// TIA Portal V17 export
// export: Created 2023-02-14T02:49:35.0431365Z, ExportSetting WithDefaults, DisplayName Totally Integrated Automation Portal, DisplayVersion V17, DisplayName TIA Portal Openness, DisplayVersion V17, DisplayName TIA Portal Teamcenter Gateway, DisplayVersion V17, DisplayName TIA Portal Version Control Interface, DisplayVersion V17, DisplayName SINAMICS Startdrive Advanced, DisplayVersion V17, DisplayName SINAMICS Startdrive G130, G150, S120, S150, SINAMICS MV, S210, DisplayVersion V17, DisplayName SINAMICS Startdrive G110M, G120, G120C, G120D, G120P, G115D, DisplayVersion V17, DisplayName STEP 7 Professional, DisplayVersion V17, DisplayName STEP 7 Safety, DisplayVersion V17, DisplayName WinCC Professional, DisplayVersion V17
FUNCTION_BLOCK "IO Valve T09 Garlic"   // FB309, LAD
{ S7_Optimized_Access := 'FALSE' }
VERSION : 0.1
// stored: AutoNumber false, IsIECCheckEnabled false, SetENOAutomatically false, UDAEnableTagReadback false
   VAR_INPUT
      lock : Bool;
      Init : Bool;
      testing : Bool;
      Reset : Bool;
   END_VAR
   VAR
      "AV-09.01" { S7_SetPoint := 'True'} : "Valve";   // AUTO BUTTERFLY VALVE INLET PROCESS WATER TO BFT GARLIC T-09.00
      "AV-09.02" { S7_SetPoint := 'True'} : "Valve";   // AUTO BUTTERFLY VALVE CIP SUPPLY TO BFT GARLIC T-09.00
      "AV-09.03" { S7_SetPoint := 'True'} : "Valve";   // AUTO BUTTERFLY VALVE OUTLET PRODUCT FROM BFT GARLIC T-09.00
      "AV-09.04" { S7_SetPoint := 'True'} : "Valve";   // AUTO BUTTERFLY VALVE CIP SUPPLY TO BFT GARLIC T-09.00
      "AV-09.05" { S7_SetPoint := 'True'} : "Valve";   // AUTO BUTTERFLY VALVE CIP SUPPLY TO BFT GARLIC T-09.00
      "AV-09.06" { S7_SetPoint := 'True'} : "Valve";   // AUTO BUTTERFLY VALVE DRAIN MONO PUMP P-09.01
      "AV-09.07" { S7_SetPoint := 'True'} : "Valve";   // AUTO BUTTERFLY VALVE INLET VINEGAR FROM T-10.00 TO BLENDING TANK T-20.00
      "AV-09.08" { S7_SetPoint := 'True'} : "Valve";
      "AV-09.09" { S7_SetPoint := 'True'} : "Valve";
      "AV-09.10" { S7_SetPoint := 'True'} : "Valve";
      "AV-09.11" { S7_SetPoint := 'True'} : "Valve";
      "AV-09.12" { S7_SetPoint := 'True'} : "Valve";
      "AV-09.13" { S7_SetPoint := 'True'} : "Valve";
      "AV-09.14" { S7_SetPoint := 'True'} : "Valve";
      "AV-09.15" { S7_SetPoint := 'True'} : "Valve";
   END_VAR
BEGIN

REGION Network 1 (SCL): FB OPEN and CLOSE
   IF #testing THEN
       // Statement section IF
       #"AV-09.01".FB_OPEN := #"AV-09.01".QCMD_OP;
       #"AV-09.01".FB_CLOSE := NOT #"AV-09.01".QCMD_OP;
       #"AV-09.02".FB_OPEN := #"AV-09.02".QCMD_OP;
       #"AV-09.02".FB_CLOSE := NOT #"AV-09.02".QCMD_OP;
       #"AV-09.03".FB_OPEN := #"AV-09.03".QCMD_OP;
       #"AV-09.03".FB_CLOSE := NOT #"AV-09.03".QCMD_OP;
       #"AV-09.04".FB_OPEN := #"AV-09.04".QCMD_OP;
       #"AV-09.04".FB_CLOSE := NOT #"AV-09.04".QCMD_OP;
       #"AV-09.05".FB_OPEN := #"AV-09.05".QCMD_OP;
       #"AV-09.05".FB_CLOSE := NOT #"AV-09.05".QCMD_OP;
       #"AV-09.06".FB_OPEN := #"AV-09.06".QCMD_OP;
       #"AV-09.06".FB_CLOSE := NOT #"AV-09.06".QCMD_OP;
       #"AV-09.07".FB_OPEN := #"AV-09.07".QCMD_OP;
       #"AV-09.07".FB_CLOSE := NOT #"AV-09.07".QCMD_OP;
       #"AV-09.08".FB_OPEN := #"AV-09.08".QCMD_OP;
       #"AV-09.08".FB_CLOSE := NOT #"AV-09.08".QCMD_OP;
       #"AV-09.09".FB_OPEN := #"AV-09.09".QCMD_OP;
       #"AV-09.09".FB_CLOSE := NOT #"AV-09.09".QCMD_OP;
       #"AV-09.10".FB_OPEN := #"AV-09.10".QCMD_OP;
       #"AV-09.10".FB_CLOSE := NOT #"AV-09.10".QCMD_OP;
       #"AV-09.11".FB_OPEN := #"AV-09.11".QCMD_OP;
       #"AV-09.11".FB_CLOSE := NOT #"AV-09.11".QCMD_OP;
       #"AV-09.12".FB_OPEN := #"AV-09.12".QCMD_OP;
       #"AV-09.12".FB_CLOSE := NOT #"AV-09.12".QCMD_OP;
       #"AV-09.13".FB_OPEN := #"AV-09.13".QCMD_OP;
       #"AV-09.13".FB_CLOSE := NOT #"AV-09.13".QCMD_OP;
       #"AV-09.14".FB_OPEN := #"AV-09.14".QCMD_OP;
       #"AV-09.14".FB_CLOSE := NOT #"AV-09.14".QCMD_OP;
       #"AV-09.15".FB_OPEN := #"AV-09.15".QCMD_OP;
       #"AV-09.15".FB_CLOSE := NOT #"AV-09.15".QCMD_OP;
   ELSE
       // Statement section ELSE
       #"AV-09.01".FB_OPEN := NOT "ZSC-09.01";
       #"AV-09.01".FB_CLOSE := "ZSC-09.01";
       #"AV-09.02".FB_OPEN := NOT "ZSC-09.02";
       #"AV-09.02".FB_CLOSE := "ZSC-09.02";
       #"AV-09.03".FB_OPEN := NOT "ZSC-09.03";
       #"AV-09.03".FB_CLOSE := "ZSC-09.03";
       #"AV-09.04".FB_OPEN := NOT "ZSC-09.04";
       #"AV-09.04".FB_CLOSE := "ZSC-09.04";
       #"AV-09.05".FB_OPEN := NOT "ZSC-09.05";
       #"AV-09.05".FB_CLOSE := "ZSC-09.05";
       #"AV-09.06".FB_OPEN := #"AV-09.06".QCMD_OP;
       #"AV-09.06".FB_CLOSE := NOT #"AV-09.06".QCMD_OP;
       #"AV-09.07".FB_OPEN := #"AV-09.07".QCMD_OP;
       #"AV-09.07".FB_CLOSE := NOT #"AV-09.07".QCMD_OP;
       #"AV-09.08".FB_OPEN := #"AV-09.08".QCMD_OP;
       #"AV-09.08".FB_CLOSE := NOT #"AV-09.08".QCMD_OP;
       #"AV-09.09".FB_OPEN := #"AV-09.09".QCMD_OP;
       #"AV-09.09".FB_CLOSE := NOT #"AV-09.09".QCMD_OP;
       #"AV-09.10".FB_OPEN := #"AV-09.10".QCMD_OP;
       #"AV-09.10".FB_CLOSE := NOT #"AV-09.10".QCMD_OP;
       #"AV-09.11".FB_OPEN := NOT "ZSC-09.11";
       #"AV-09.11".FB_CLOSE := "ZSC-09.11";
       #"AV-09.12".FB_OPEN := NOT "ZSC-09.12";
       #"AV-09.12".FB_CLOSE := "ZSC-09.12";
       #"AV-09.13".FB_OPEN := NOT "ZSC-09.13";
       #"AV-09.13".FB_CLOSE := "ZSC-09.13";
       #"AV-09.14".FB_OPEN := #"AV-09.14".QCMD_OP;
       #"AV-09.14".FB_CLOSE := NOT #"AV-09.14".QCMD_OP;
       #"AV-09.15".FB_OPEN := #"AV-09.15".QCMD_OP;
       #"AV-09.15".FB_CLOSE := NOT #"AV-09.15".QCMD_OP;
   END_IF;
END_REGION

NETWORK
TITLE = FB Monitoring Time
// FB OPEN Time
      L     t#20s;
      T     #"AV-09.01".MON_T;
      T     #"AV-09.02".MON_T;
      T     #"AV-09.03".MON_T;
      T     #"AV-09.04".MON_T;
      T     #"AV-09.05".MON_T;
      T     #"AV-09.06".MON_T;
      T     #"AV-09.07".MON_T;
      T     #"AV-09.08".MON_T;
      T     #"AV-09.09".MON_T;
      T     #"AV-09.10".MON_T;
      T     #"AV-09.11".MON_T;
      T     #"AV-09.12".MON_T;
      T     #"AV-09.13".MON_T;
      T     #"AV-09.14".MON_T;
      T     #"AV-09.15".MON_T;
// FB CLOSE Time
      L     t#20s;
      T     #"AV-09.01".MON_T_CLOSE;
      T     #"AV-09.02".MON_T_CLOSE;
      T     #"AV-09.03".MON_T_CLOSE;
      T     #"AV-09.04".MON_T_CLOSE;
      T     #"AV-09.05".MON_T_CLOSE;
      T     #"AV-09.06".MON_T_CLOSE;
      T     #"AV-09.07".MON_T_CLOSE;
      T     #"AV-09.08".MON_T_CLOSE;
      T     #"AV-09.09".MON_T_CLOSE;
      T     #"AV-09.10".MON_T_CLOSE;
      T     #"AV-09.11".MON_T_CLOSE;
      T     #"AV-09.12".MON_T_CLOSE;
      T     #"AV-09.13".MON_T_CLOSE;
      T     #"AV-09.14".MON_T_CLOSE;
      T     #"AV-09.15".MON_T_CLOSE;

REGION Network 3: AV-09.01 w ZSC
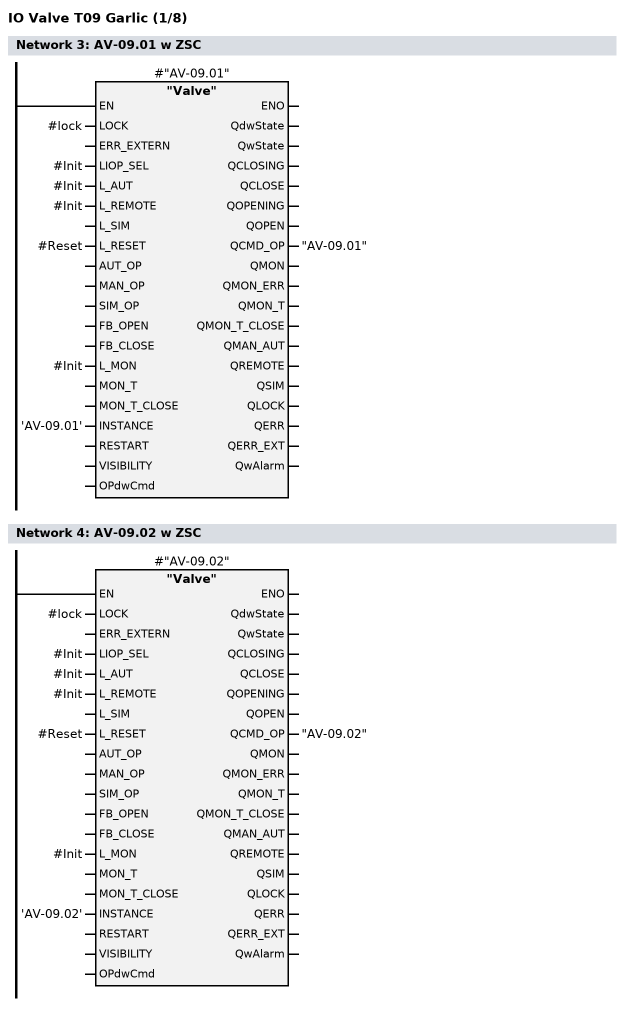
   RUNG wire#powerrail
      #"AV-09.01"(LOCK := #lock, ERR_EXTERN :=, LIOP_SEL := #Init, L_AUT := #Init, L_REMOTE := #Init, L_SIM :=, L_RESET := #Reset, AUT_OP :=, MAN_OP :=, SIM_OP :=, FB_OPEN :=, FB_CLOSE :=, L_MON := #Init, MON_T :=, MON_T_CLOSE :=, INSTANCE := 'AV-09.01', RESTART :=, VISIBILITY :=, OPdwCmd :=, QdwState =>, QwState =>, QCLOSING =>, QCLOSE =>, QOPENING =>, QOPEN =>, QCMD_OP => "AV-09.01", QMON =>, QMON_ERR =>, QMON_T =>, QMON_T_CLOSE =>, QMAN_AUT =>, QREMOTE =>, QSIM =>, QLOCK =>, QERR =>, QERR_EXT =>, QwAlarm =>)
   END_RUNG
   // the same network as SCL:
   #"AV-09.01"(LOCK := #lock,   // "Valve"
               LIOP_SEL := #Init,
               L_AUT := #Init,
               L_REMOTE := #Init,
               L_RESET := #Reset,
               L_MON := #Init,
               INSTANCE := 'AV-09.01',
               QCMD_OP => "AV-09.01");
END_REGION

REGION Network 4: AV-09.02 w ZSC
   RUNG wire#powerrail
      #"AV-09.02"(LOCK := #lock, ERR_EXTERN :=, LIOP_SEL := #Init, L_AUT := #Init, L_REMOTE := #Init, L_SIM :=, L_RESET := #Reset, AUT_OP :=, MAN_OP :=, SIM_OP :=, FB_OPEN :=, FB_CLOSE :=, L_MON := #Init, MON_T :=, MON_T_CLOSE :=, INSTANCE := 'AV-09.02', RESTART :=, VISIBILITY :=, OPdwCmd :=, QdwState =>, QwState =>, QCLOSING =>, QCLOSE =>, QOPENING =>, QOPEN =>, QCMD_OP => "AV-09.02", QMON =>, QMON_ERR =>, QMON_T =>, QMON_T_CLOSE =>, QMAN_AUT =>, QREMOTE =>, QSIM =>, QLOCK =>, QERR =>, QERR_EXT =>, QwAlarm =>)
   END_RUNG
   // the same network as SCL:
   #"AV-09.02"(LOCK := #lock,   // "Valve"
               LIOP_SEL := #Init,
               L_AUT := #Init,
               L_REMOTE := #Init,
               L_RESET := #Reset,
               L_MON := #Init,
               INSTANCE := 'AV-09.02',
               QCMD_OP => "AV-09.02");
END_REGION

REGION Network 5: AV-09.03 w ZSC
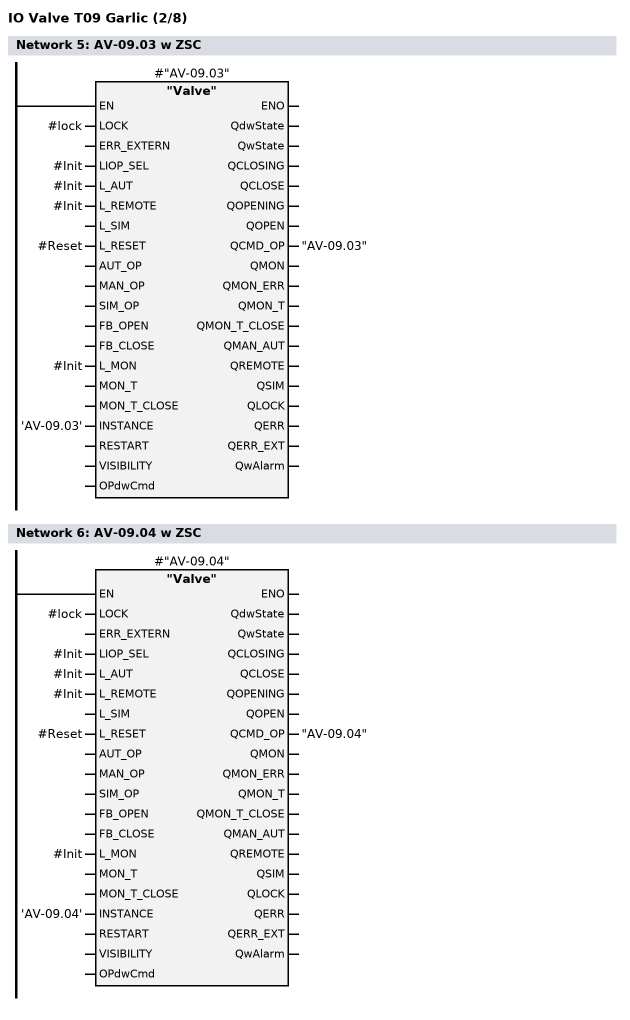
   RUNG wire#powerrail
      #"AV-09.03"(LOCK := #lock, ERR_EXTERN :=, LIOP_SEL := #Init, L_AUT := #Init, L_REMOTE := #Init, L_SIM :=, L_RESET := #Reset, AUT_OP :=, MAN_OP :=, SIM_OP :=, FB_OPEN :=, FB_CLOSE :=, L_MON := #Init, MON_T :=, MON_T_CLOSE :=, INSTANCE := 'AV-09.03', RESTART :=, VISIBILITY :=, OPdwCmd :=, QdwState =>, QwState =>, QCLOSING =>, QCLOSE =>, QOPENING =>, QOPEN =>, QCMD_OP => "AV-09.03", QMON =>, QMON_ERR =>, QMON_T =>, QMON_T_CLOSE =>, QMAN_AUT =>, QREMOTE =>, QSIM =>, QLOCK =>, QERR =>, QERR_EXT =>, QwAlarm =>)
   END_RUNG
   // the same network as SCL:
   #"AV-09.03"(LOCK := #lock,   // "Valve"
               LIOP_SEL := #Init,
               L_AUT := #Init,
               L_REMOTE := #Init,
               L_RESET := #Reset,
               L_MON := #Init,
               INSTANCE := 'AV-09.03',
               QCMD_OP => "AV-09.03");
END_REGION

REGION Network 6: AV-09.04 w ZSC
   RUNG wire#powerrail
      #"AV-09.04"(LOCK := #lock, ERR_EXTERN :=, LIOP_SEL := #Init, L_AUT := #Init, L_REMOTE := #Init, L_SIM :=, L_RESET := #Reset, AUT_OP :=, MAN_OP :=, SIM_OP :=, FB_OPEN :=, FB_CLOSE :=, L_MON := #Init, MON_T :=, MON_T_CLOSE :=, INSTANCE := 'AV-09.04', RESTART :=, VISIBILITY :=, OPdwCmd :=, QdwState =>, QwState =>, QCLOSING =>, QCLOSE =>, QOPENING =>, QOPEN =>, QCMD_OP => "AV-09.04", QMON =>, QMON_ERR =>, QMON_T =>, QMON_T_CLOSE =>, QMAN_AUT =>, QREMOTE =>, QSIM =>, QLOCK =>, QERR =>, QERR_EXT =>, QwAlarm =>)
   END_RUNG
   // the same network as SCL:
   #"AV-09.04"(LOCK := #lock,   // "Valve"
               LIOP_SEL := #Init,
               L_AUT := #Init,
               L_REMOTE := #Init,
               L_RESET := #Reset,
               L_MON := #Init,
               INSTANCE := 'AV-09.04',
               QCMD_OP => "AV-09.04");
END_REGION

REGION Network 7: AV-09.05 w ZSC
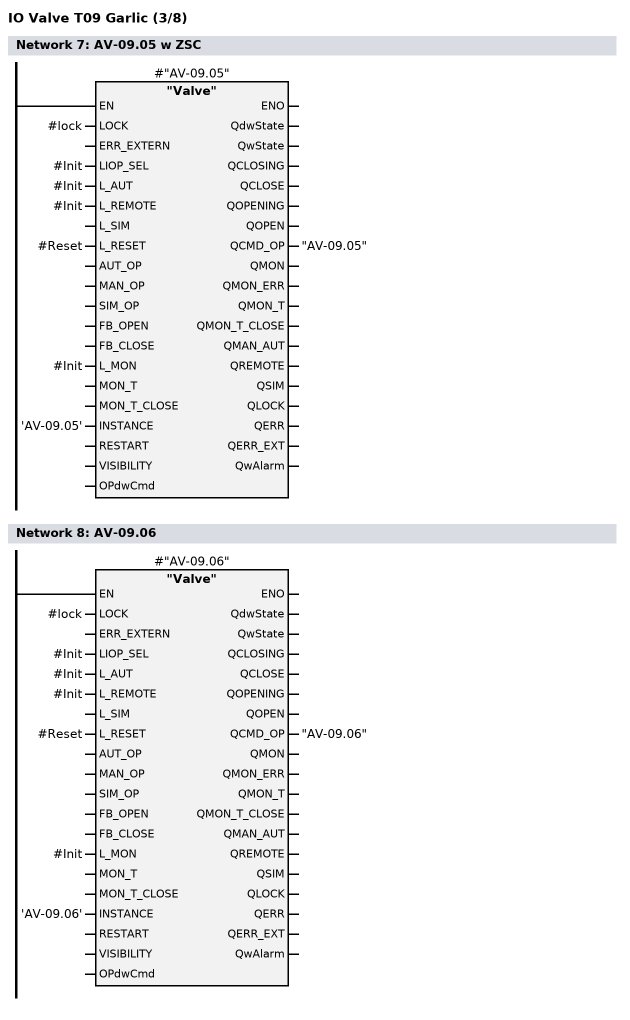
   RUNG wire#powerrail
      #"AV-09.05"(LOCK := #lock, ERR_EXTERN :=, LIOP_SEL := #Init, L_AUT := #Init, L_REMOTE := #Init, L_SIM :=, L_RESET := #Reset, AUT_OP :=, MAN_OP :=, SIM_OP :=, FB_OPEN :=, FB_CLOSE :=, L_MON := #Init, MON_T :=, MON_T_CLOSE :=, INSTANCE := 'AV-09.05', RESTART :=, VISIBILITY :=, OPdwCmd :=, QdwState =>, QwState =>, QCLOSING =>, QCLOSE =>, QOPENING =>, QOPEN =>, QCMD_OP => "AV-09.05", QMON =>, QMON_ERR =>, QMON_T =>, QMON_T_CLOSE =>, QMAN_AUT =>, QREMOTE =>, QSIM =>, QLOCK =>, QERR =>, QERR_EXT =>, QwAlarm =>)
   END_RUNG
   // the same network as SCL:
   #"AV-09.05"(LOCK := #lock,   // "Valve"
               LIOP_SEL := #Init,
               L_AUT := #Init,
               L_REMOTE := #Init,
               L_RESET := #Reset,
               L_MON := #Init,
               INSTANCE := 'AV-09.05',
               QCMD_OP => "AV-09.05");
END_REGION

REGION Network 8: AV-09.06
   RUNG wire#powerrail
      #"AV-09.06"(LOCK := #lock, ERR_EXTERN :=, LIOP_SEL := #Init, L_AUT := #Init, L_REMOTE := #Init, L_SIM :=, L_RESET := #Reset, AUT_OP :=, MAN_OP :=, SIM_OP :=, FB_OPEN :=, FB_CLOSE :=, L_MON := #Init, MON_T :=, MON_T_CLOSE :=, INSTANCE := 'AV-09.06', RESTART :=, VISIBILITY :=, OPdwCmd :=, QdwState =>, QwState =>, QCLOSING =>, QCLOSE =>, QOPENING =>, QOPEN =>, QCMD_OP => "AV-09.06", QMON =>, QMON_ERR =>, QMON_T =>, QMON_T_CLOSE =>, QMAN_AUT =>, QREMOTE =>, QSIM =>, QLOCK =>, QERR =>, QERR_EXT =>, QwAlarm =>)
   END_RUNG
   // the same network as SCL:
   #"AV-09.06"(LOCK := #lock,   // "Valve"
               LIOP_SEL := #Init,
               L_AUT := #Init,
               L_REMOTE := #Init,
               L_RESET := #Reset,
               L_MON := #Init,
               INSTANCE := 'AV-09.06',
               QCMD_OP => "AV-09.06");
END_REGION

REGION Network 9: AV-09.07
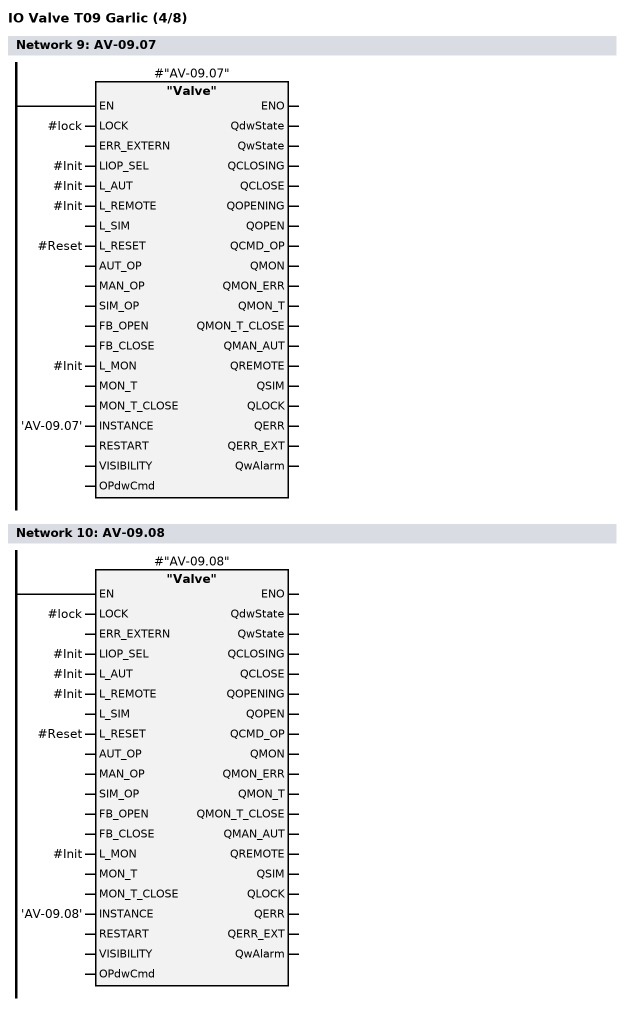
   RUNG wire#powerrail
      #"AV-09.07"(LOCK := #lock, ERR_EXTERN :=, LIOP_SEL := #Init, L_AUT := #Init, L_REMOTE := #Init, L_SIM :=, L_RESET := #Reset, AUT_OP :=, MAN_OP :=, SIM_OP :=, FB_OPEN :=, FB_CLOSE :=, L_MON := #Init, MON_T :=, MON_T_CLOSE :=, INSTANCE := 'AV-09.07', RESTART :=, VISIBILITY :=, OPdwCmd :=, QdwState =>, QwState =>, QCLOSING =>, QCLOSE =>, QOPENING =>, QOPEN =>, QCMD_OP =>, QMON =>, QMON_ERR =>, QMON_T =>, QMON_T_CLOSE =>, QMAN_AUT =>, QREMOTE =>, QSIM =>, QLOCK =>, QERR =>, QERR_EXT =>, QwAlarm =>)
   END_RUNG
   // the same network as SCL:
   #"AV-09.07"(LOCK := #lock,   // "Valve"
               LIOP_SEL := #Init,
               L_AUT := #Init,
               L_REMOTE := #Init,
               L_RESET := #Reset,
               L_MON := #Init,
               INSTANCE := 'AV-09.07');
END_REGION

REGION Network 10: AV-09.08
   RUNG wire#powerrail
      #"AV-09.08"(LOCK := #lock, ERR_EXTERN :=, LIOP_SEL := #Init, L_AUT := #Init, L_REMOTE := #Init, L_SIM :=, L_RESET := #Reset, AUT_OP :=, MAN_OP :=, SIM_OP :=, FB_OPEN :=, FB_CLOSE :=, L_MON := #Init, MON_T :=, MON_T_CLOSE :=, INSTANCE := 'AV-09.08', RESTART :=, VISIBILITY :=, OPdwCmd :=, QdwState =>, QwState =>, QCLOSING =>, QCLOSE =>, QOPENING =>, QOPEN =>, QCMD_OP =>, QMON =>, QMON_ERR =>, QMON_T =>, QMON_T_CLOSE =>, QMAN_AUT =>, QREMOTE =>, QSIM =>, QLOCK =>, QERR =>, QERR_EXT =>, QwAlarm =>)
   END_RUNG
   // the same network as SCL:
   #"AV-09.08"(LOCK := #lock,   // "Valve"
               LIOP_SEL := #Init,
               L_AUT := #Init,
               L_REMOTE := #Init,
               L_RESET := #Reset,
               L_MON := #Init,
               INSTANCE := 'AV-09.08');
END_REGION

REGION Network 11: AV-09.09
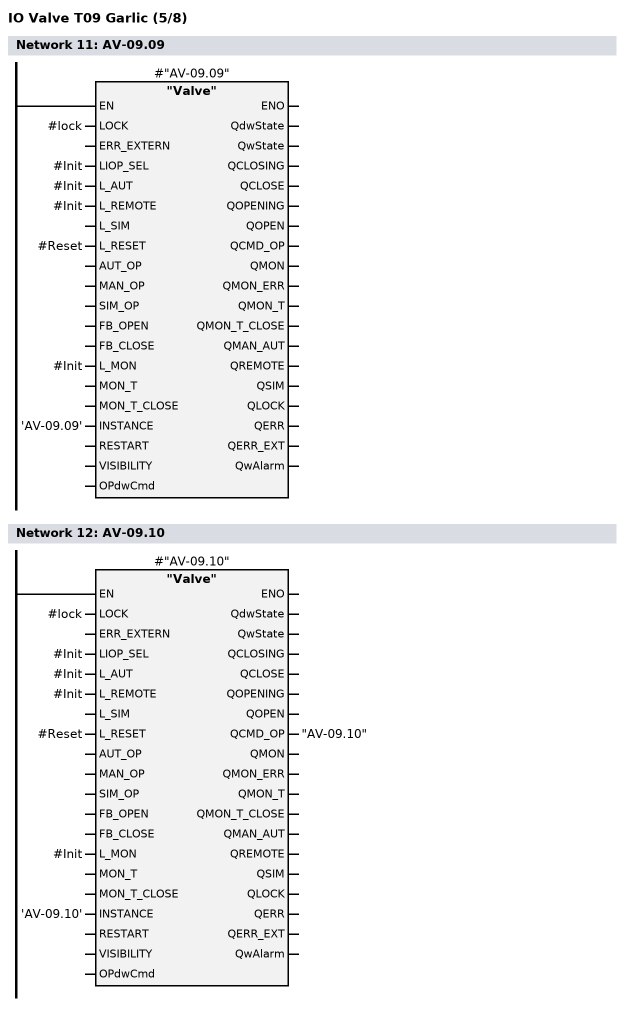
   RUNG wire#powerrail
      #"AV-09.09"(LOCK := #lock, ERR_EXTERN :=, LIOP_SEL := #Init, L_AUT := #Init, L_REMOTE := #Init, L_SIM :=, L_RESET := #Reset, AUT_OP :=, MAN_OP :=, SIM_OP :=, FB_OPEN :=, FB_CLOSE :=, L_MON := #Init, MON_T :=, MON_T_CLOSE :=, INSTANCE := 'AV-09.09', RESTART :=, VISIBILITY :=, OPdwCmd :=, QdwState =>, QwState =>, QCLOSING =>, QCLOSE =>, QOPENING =>, QOPEN =>, QCMD_OP =>, QMON =>, QMON_ERR =>, QMON_T =>, QMON_T_CLOSE =>, QMAN_AUT =>, QREMOTE =>, QSIM =>, QLOCK =>, QERR =>, QERR_EXT =>, QwAlarm =>)
   END_RUNG
   // the same network as SCL:
   #"AV-09.09"(LOCK := #lock,   // "Valve"
               LIOP_SEL := #Init,
               L_AUT := #Init,
               L_REMOTE := #Init,
               L_RESET := #Reset,
               L_MON := #Init,
               INSTANCE := 'AV-09.09');
END_REGION

REGION Network 12: AV-09.10
   RUNG wire#powerrail
      #"AV-09.10"(LOCK := #lock, ERR_EXTERN :=, LIOP_SEL := #Init, L_AUT := #Init, L_REMOTE := #Init, L_SIM :=, L_RESET := #Reset, AUT_OP :=, MAN_OP :=, SIM_OP :=, FB_OPEN :=, FB_CLOSE :=, L_MON := #Init, MON_T :=, MON_T_CLOSE :=, INSTANCE := 'AV-09.10', RESTART :=, VISIBILITY :=, OPdwCmd :=, QdwState =>, QwState =>, QCLOSING =>, QCLOSE =>, QOPENING =>, QOPEN =>, QCMD_OP => "AV-09.10", QMON =>, QMON_ERR =>, QMON_T =>, QMON_T_CLOSE =>, QMAN_AUT =>, QREMOTE =>, QSIM =>, QLOCK =>, QERR =>, QERR_EXT =>, QwAlarm =>)
   END_RUNG
   // the same network as SCL:
   #"AV-09.10"(LOCK := #lock,   // "Valve"
               LIOP_SEL := #Init,
               L_AUT := #Init,
               L_REMOTE := #Init,
               L_RESET := #Reset,
               L_MON := #Init,
               INSTANCE := 'AV-09.10',
               QCMD_OP => "AV-09.10");
END_REGION

REGION Network 13: AV-09.11 w ZSC
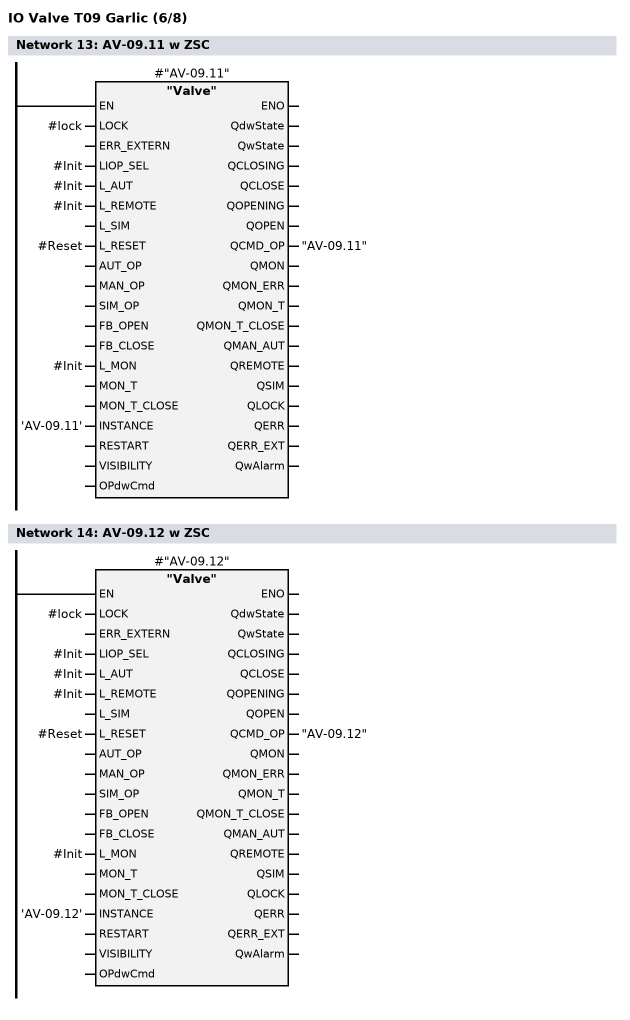
   RUNG wire#powerrail
      #"AV-09.11"(LOCK := #lock, ERR_EXTERN :=, LIOP_SEL := #Init, L_AUT := #Init, L_REMOTE := #Init, L_SIM :=, L_RESET := #Reset, AUT_OP :=, MAN_OP :=, SIM_OP :=, FB_OPEN :=, FB_CLOSE :=, L_MON := #Init, MON_T :=, MON_T_CLOSE :=, INSTANCE := 'AV-09.11', RESTART :=, VISIBILITY :=, OPdwCmd :=, QdwState =>, QwState =>, QCLOSING =>, QCLOSE =>, QOPENING =>, QOPEN =>, QCMD_OP => "AV-09.11", QMON =>, QMON_ERR =>, QMON_T =>, QMON_T_CLOSE =>, QMAN_AUT =>, QREMOTE =>, QSIM =>, QLOCK =>, QERR =>, QERR_EXT =>, QwAlarm =>)
   END_RUNG
   // the same network as SCL:
   #"AV-09.11"(LOCK := #lock,   // "Valve"
               LIOP_SEL := #Init,
               L_AUT := #Init,
               L_REMOTE := #Init,
               L_RESET := #Reset,
               L_MON := #Init,
               INSTANCE := 'AV-09.11',
               QCMD_OP => "AV-09.11");
END_REGION

REGION Network 14: AV-09.12 w ZSC
   RUNG wire#powerrail
      #"AV-09.12"(LOCK := #lock, ERR_EXTERN :=, LIOP_SEL := #Init, L_AUT := #Init, L_REMOTE := #Init, L_SIM :=, L_RESET := #Reset, AUT_OP :=, MAN_OP :=, SIM_OP :=, FB_OPEN :=, FB_CLOSE :=, L_MON := #Init, MON_T :=, MON_T_CLOSE :=, INSTANCE := 'AV-09.12', RESTART :=, VISIBILITY :=, OPdwCmd :=, QdwState =>, QwState =>, QCLOSING =>, QCLOSE =>, QOPENING =>, QOPEN =>, QCMD_OP => "AV-09.12", QMON =>, QMON_ERR =>, QMON_T =>, QMON_T_CLOSE =>, QMAN_AUT =>, QREMOTE =>, QSIM =>, QLOCK =>, QERR =>, QERR_EXT =>, QwAlarm =>)
   END_RUNG
   // the same network as SCL:
   #"AV-09.12"(LOCK := #lock,   // "Valve"
               LIOP_SEL := #Init,
               L_AUT := #Init,
               L_REMOTE := #Init,
               L_RESET := #Reset,
               L_MON := #Init,
               INSTANCE := 'AV-09.12',
               QCMD_OP => "AV-09.12");
END_REGION

REGION Network 15: AV-09.13 w ZSC
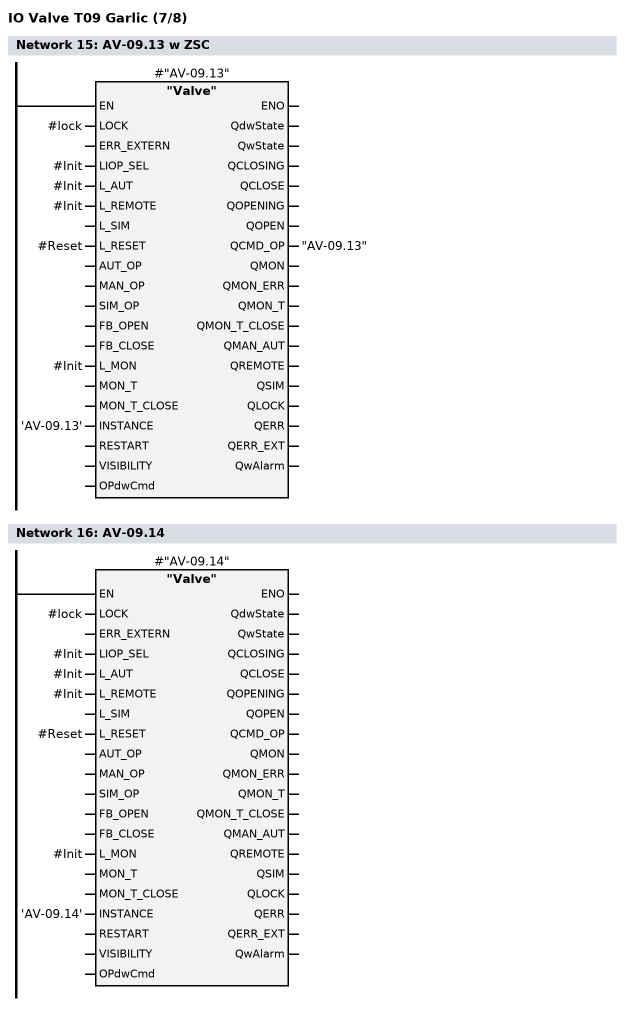
   RUNG wire#powerrail
      #"AV-09.13"(LOCK := #lock, ERR_EXTERN :=, LIOP_SEL := #Init, L_AUT := #Init, L_REMOTE := #Init, L_SIM :=, L_RESET := #Reset, AUT_OP :=, MAN_OP :=, SIM_OP :=, FB_OPEN :=, FB_CLOSE :=, L_MON := #Init, MON_T :=, MON_T_CLOSE :=, INSTANCE := 'AV-09.13', RESTART :=, VISIBILITY :=, OPdwCmd :=, QdwState =>, QwState =>, QCLOSING =>, QCLOSE =>, QOPENING =>, QOPEN =>, QCMD_OP => "AV-09.13", QMON =>, QMON_ERR =>, QMON_T =>, QMON_T_CLOSE =>, QMAN_AUT =>, QREMOTE =>, QSIM =>, QLOCK =>, QERR =>, QERR_EXT =>, QwAlarm =>)
   END_RUNG
   // the same network as SCL:
   #"AV-09.13"(LOCK := #lock,   // "Valve"
               LIOP_SEL := #Init,
               L_AUT := #Init,
               L_REMOTE := #Init,
               L_RESET := #Reset,
               L_MON := #Init,
               INSTANCE := 'AV-09.13',
               QCMD_OP => "AV-09.13");
END_REGION

REGION Network 16: AV-09.14
   RUNG wire#powerrail
      #"AV-09.14"(LOCK := #lock, ERR_EXTERN :=, LIOP_SEL := #Init, L_AUT := #Init, L_REMOTE := #Init, L_SIM :=, L_RESET := #Reset, AUT_OP :=, MAN_OP :=, SIM_OP :=, FB_OPEN :=, FB_CLOSE :=, L_MON := #Init, MON_T :=, MON_T_CLOSE :=, INSTANCE := 'AV-09.14', RESTART :=, VISIBILITY :=, OPdwCmd :=, QdwState =>, QwState =>, QCLOSING =>, QCLOSE =>, QOPENING =>, QOPEN =>, QCMD_OP =>, QMON =>, QMON_ERR =>, QMON_T =>, QMON_T_CLOSE =>, QMAN_AUT =>, QREMOTE =>, QSIM =>, QLOCK =>, QERR =>, QERR_EXT =>, QwAlarm =>)
   END_RUNG
   // the same network as SCL:
   #"AV-09.14"(LOCK := #lock,   // "Valve"
               LIOP_SEL := #Init,
               L_AUT := #Init,
               L_REMOTE := #Init,
               L_RESET := #Reset,
               L_MON := #Init,
               INSTANCE := 'AV-09.14');
END_REGION

REGION Network 17: AV-09.15
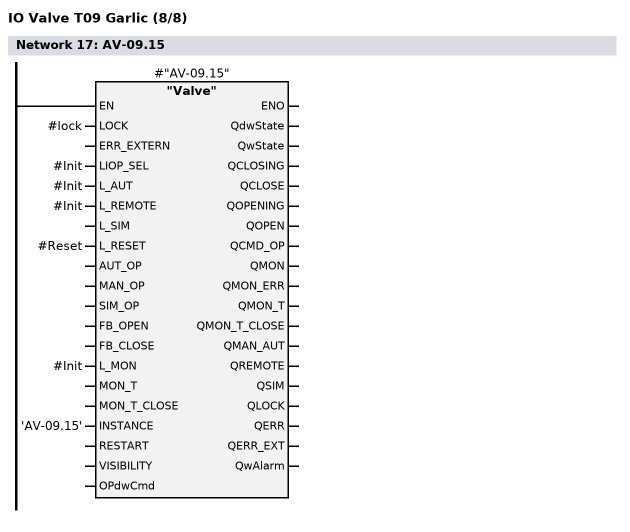
   RUNG wire#powerrail
      #"AV-09.15"(LOCK := #lock, ERR_EXTERN :=, LIOP_SEL := #Init, L_AUT := #Init, L_REMOTE := #Init, L_SIM :=, L_RESET := #Reset, AUT_OP :=, MAN_OP :=, SIM_OP :=, FB_OPEN :=, FB_CLOSE :=, L_MON := #Init, MON_T :=, MON_T_CLOSE :=, INSTANCE := 'AV-09.15', RESTART :=, VISIBILITY :=, OPdwCmd :=, QdwState =>, QwState =>, QCLOSING =>, QCLOSE =>, QOPENING =>, QOPEN =>, QCMD_OP =>, QMON =>, QMON_ERR =>, QMON_T =>, QMON_T_CLOSE =>, QMAN_AUT =>, QREMOTE =>, QSIM =>, QLOCK =>, QERR =>, QERR_EXT =>, QwAlarm =>)
   END_RUNG
   // the same network as SCL:
   #"AV-09.15"(LOCK := #lock,   // "Valve"
               LIOP_SEL := #Init,
               L_AUT := #Init,
               L_REMOTE := #Init,
               L_RESET := #Reset,
               L_MON := #Init,
               INSTANCE := 'AV-09.15');
END_REGION
END_FUNCTION_BLOCK
